LIN {X 0,Y 197.414,Z 518.474,A -85,B 0,C 180,E1 1852.576,E2 1852.576} C_VEL
LIN {X 0,Y 195.678,Z 514.647,A -85,B 0,C 180,E1 1845.984,E2 1845.984} C_VEL
LIN {X 0,Y 194.931,Z 514.01,A -85,B 0,C 180,E1 1839.244,E2 1839.244} C_VEL
LIN {X 0,Y 195.748,Z 514.716,A -85,B 0,C 180,E1 1832.022,E2 1832.022} C_VEL
LIN {X 0,Y 197.692,Z 519.438,A -85,B 0,C 180,E1 1824.497,E2 1824.497} C_VEL
LIN {X 0,Y 199.785,Z 523.662,A -85,B 0,C 180,E1 1819.811,E2 1819.811} C_VEL
LIN {X 0,Y 202.216,Z 528.549,A -85,B 0,C 180,E1 1815.605,E2 1815.605} C_VEL
LIN {X 0,Y 190.643,Z 578.863,A -85,B 0,C 180,E1 1815.121,E2 1815.121} C_VEL
LIN {X 0,Y 183.364,Z 602.487,A -85,B 0,C 180,E1 1814.882,E2 1814.882} C_VEL
LIN {X 0,Y 173.66,Z 626.987,A -85,B 0,C 180,E1 1814.716,E2 1814.716} C_VEL
LIN {X 0,Y 162.076,Z 650.907,A -85,B 0,C 180,E1 1814.426,E2 1814.426} C_VEL
LIN {X 0,Y 149.405,Z 672.786,A -85,B 0,C 180,E1 1813.999,E2 1813.999} C_VEL
LIN {X 0,Y 135.148,Z 693.676,A -85,B 0,C 180,E1 1813.399,E2 1813.399} C_VEL
LIN {X 0,Y 120.37,Z 712.234,A -85,B 0,C 180,E1 1812.599,E2 1812.599} C_VEL
LIN {X 0,Y 104.563,Z 729.321,A -85,B 0,C 180,E1 1811.473,E2 1811.473} C_VEL
LIN {X 0,Y 87.256,Z 745.402,A -85,B 0,C 180,E1 1809.824,E2 1809.824} C_VEL
LIN {X 0,Y 69.557,Z 759.526,A -85,B 0,C 180,E1 1807.39,E2 1807.39} C_VEL
LIN {X 0,Y 52.081,Z 771.407,A -85,B 0,C 180,E1 1803.53,E2 1803.53} C_VEL
LIN {X 0,Y 34.078,Z 781.783,A -85,B 0,C 180,E1 1795.754,E2 1795.754} C_VEL
LIN {X 0,Y 17.731,Z 790.254,A -85,B 0,C 180,E1 1774.376,E2 1774.376} C_VEL
LIN {X 0,Y 11.425,Z 796.051,A -85,B 0,C 180,E1 1709.95,E2 1709.95} C_VEL
LIN {X 0,Y 11.818,Z 796.617,A -85,B 0,C 180,E1 1700.209,E2 1700.209} C_VEL
LIN {X 0,Y 14.795,Z 798.166,A -85,B 0,C 180,E1 1657.527,E2 1657.527} C_VEL
LIN {X 0,Y 9.219,Z 793.702,A -85,B 0,C 180,E1 1601.102,E2 1601.102} C_VEL
LIN {X 0,Y 18.153,Z 786.818,A -85,B 0,C 180,E1 1537.839,E2 1537.839} C_VEL
LIN {X 0,Y 35.521,Z 777.013,A -85,B 0,C 180,E1 1519.997,E2 1519.997} C_VEL
LIN {X 0,Y 54.697,Z 764.948,A -85,B 0,C 180,E1 1513.005,E2 1513.005} C_VEL
LIN {X 0,Y 72.604,Z 751.86,A -85,B 0,C 180,E1 1509.431,E2 1509.431} C_VEL
LIN {X 0,Y 90.666,Z 736.479,A -85,B 0,C 180,E1 1507.024,E2 1507.024} C_VEL
LIN {X 0,Y 107.146,Z 720.254,A -85,B 0,C 180,E1 1505.379,E2 1505.379} C_VEL
LIN {X 0,Y 123.373,Z 701.747,A -85,B 0,C 180,E1 1504.086,E2 1504.086} C_VEL
LIN {X 0,Y 132.523,Z 689.974,A -85,B 0,C 180,E1 1503.457,E2 1503.457} C_VEL
LIN {X 0,Y 136.821,Z 683.736,A -85,B 0,C 180,E1 1502.763,E2 1502.763} C_VEL
LIN {X 0,Y 146.781,Z 666.497,A -85,B 0,C 180,E1 1499.753,E2 1499.753} C_VEL
LIN {X 0,Y 150.068,Z 660.76,A -85,B 0,C 180,E1 1499.343,E2 1499.343} C_VEL
LIN {X 0,Y 162.241,Z 638.701,A -85,B 0,C 180,E1 1498.929,E2 1498.929} C_VEL
LIN {X 0,Y 172.705,Z 616.198,A -85,B 0,C 180,E1 1498.602,E2 1498.602} C_VEL
LIN {X 0,Y 182.088,Z 591.601,A -85,B 0,C 180,E1 1498.323,E2 1498.323} C_VEL
LIN {X 0,Y 189.755,Z 566.126,A -85,B 0,C 180,E1 1498.101,E2 1498.101} C_VEL
LIN {X 0,Y 197.833,Z 531.198,A -85,B 0,C 180,E1 1497.859,E2 1497.859} C_VEL
LIN {X 0,Y 195.599,Z 526.307,A -85,B 0,C 180,E1 1492.537,E2 1492.537} C_VEL
LIN {X 0,Y 193.851,Z 522.423,A -85,B 0,C 180,E1 1485.795,E2 1485.795} C_VEL
LIN {X 0,Y 193.15,Z 521.811,A -85,B 0,C 180,E1 1479.065,E2 1479.065} C_VEL
LIN {X 0,Y 193.929,Z 522.613,A -85,B 0,C 180,E1 1472.071,E2 1472.071} C_VEL
LIN {X 0,Y 195.706,Z 527.054,A -85,B 0,C 180,E1 1464.924,E2 1464.924} C_VEL
LIN {X 0,Y 197.708,Z 531.241,A -85,B 0,C 180,E1 1460.264,E2 1460.264} C_VEL
LIN {X 0,Y 198.994,Z 534.087,A -85,B 0,C 180,E1 1457.774,E2 1457.774} C_VEL
LIN {X 0,Y 188.414,Z 579.035,A -85,B 0,C 180,E1 1457.449,E2 1457.449} C_VEL
LIN {X 0,Y 181.163,Z 602.307,A -85,B 0,C 180,E1 1457.304,E2 1457.304} C_VEL
LIN {X 0,Y 171.68,Z 626.174,A -85,B 0,C 180,E1 1457.274,E2 1457.274} C_VEL
LIN {X 0,Y 160.099,Z 650.057,A -85,B 0,C 180,E1 1457.167,E2 1457.167} C_VEL
LIN {X 0,Y 147.264,Z 672.137,A -85,B 0,C 180,E1 1456.969,E2 1456.969} C_VEL
LIN {X 0,Y 133.065,Z 692.712,A -85,B 0,C 180,E1 1456.673,E2 1456.673} C_VEL
LIN {X 0,Y 118.735,Z 710.564,A -85,B 0,C 180,E1 1456.283,E2 1456.283} C_VEL
LIN {X 0,Y 102.284,Z 728.281,A -85,B 0,C 180,E1 1455.686,E2 1455.686} C_VEL
LIN {X 0,Y 84.816,Z 744.397,A -85,B 0,C 180,E1 1454.865,E2 1454.865} C_VEL
LIN {X 0,Y 67.933,Z 757.735,A -85,B 0,C 180,E1 1453.773,E2 1453.773} C_VEL
LIN {X 0,Y 50.078,Z 769.624,A -85,B 0,C 180,E1 1452.007,E2 1452.007} C_VEL
LIN {X 0,Y 30.308,Z 780.674,A -85,B 0,C 180,E1 1448.365,E2 1448.365} C_VEL
LIN {X 0,Y 12.995,Z 788.665,A -85,B 0,C 180,E1 1438.177,E2 1438.177} C_VEL
LIN {X 0,Y 4.365,Z 794.222,A -85,B 0,C 180,E1 1322.59,E2 1322.59} C_VEL
LIN {X 0,Y 4.321,Z 794.234,A -85,B 0,C 180,E1 1315.544,E2 1315.544} C_VEL
LIN {X 0,Y 8.811,Z 788.86,A -85,B 0,C 180,E1 1156.948,E2 1156.948} C_VEL
LIN {X 0,Y 27.983,Z 779.327,A -85,B 0,C 180,E1 1148.202,E2 1148.202} C_VEL
LIN {X 0,Y 46.158,Z 768.699,A -85,B 0,C 180,E1 1145.432,E2 1145.432} C_VEL
LIN {X 0,Y 65.276,Z 755.458,A -85,B 0,C 180,E1 1143.638,E2 1143.638} C_VEL
LIN {X 0,Y 83.49,Z 740.749,A -85,B 0,C 180,E1 1142.378,E2 1142.378} C_VEL
LIN {X 0,Y 100.753,Z 724.51,A -85,B 0,C 180,E1 1141.414,E2 1141.414} C_VEL
LIN {X 0,Y 116.998,Z 706.864,A -85,B 0,C 180,E1 1140.639,E2 1140.639} C_VEL
LIN {X 0,Y 132.779,Z 686.918,A -85,B 0,C 180,E1 1139.98,E2 1139.98} C_VEL
LIN {X 0,Y 146.231,Z 667.041,A -85,B 0,C 180,E1 1139.476,E2 1139.476} C_VEL
LIN {X 0,Y 150.068,Z 660.76,A -85,B 0,C 180,E1 1139.343,E2 1139.343} C_VEL
LIN {X 0,Y 153.729,Z 654.207,A -85,B 0,C 180,E1 1138.842,E2 1138.842} C_VEL
LIN {X 0,Y 162.215,Z 635.803,A -85,B 0,C 180,E1 1136.382,E2 1136.382} C_VEL
LIN {X 0,Y 165.007,Z 629.769,A -85,B 0,C 180,E1 1136.081,E2 1136.081} C_VEL
LIN {X 0,Y 175.459,Z 605.484,A -85,B 0,C 180,E1 1135.917,E2 1135.917} C_VEL
LIN {X 0,Y 184.182,Z 580.142,A -85,B 0,C 180,E1 1135.777,E2 1135.777} C_VEL
LIN {X 0,Y 191.07,Z 554.146,A -85,B 0,C 180,E1 1135.68,E2 1135.68} C_VEL
LIN {X 0,Y 194.927,Z 536.894,A -85,B 0,C 180,E1 1135.566,E2 1135.566} C_VEL
LIN {X 0,Y 193.45,Z 533.708,A -85,B 0,C 180,E1 1131.672,E2 1131.672} C_VEL
LIN {X 0,Y 192.007,Z 530.188,A -85,B 0,C 180,E1 1125.506,E2 1125.506} C_VEL
LIN {X 0,Y 191.371,Z 529.622,A -85,B 0,C 180,E1 1118.82,E2 1118.82} C_VEL
LIN {X 0,Y 192.091,Z 530.439,A -85,B 0,C 180,E1 1112.238,E2 1112.238} C_VEL
LIN {X 0,Y 193.731,Z 534.669,A -85,B 0,C 180,E1 1105.359,E2 1105.359} C_VEL
LIN {X 0,Y 195.639,Z 538.806,A -85,B 0,C 180,E1 1100.739,E2 1100.739} C_VEL
LIN {X 0,Y 195.909,Z 539.823,A -85,B 0,C 180,E1 1100.007,E2 1100.007} C_VEL
LIN {X 0,Y 186.521,Z 579.131,A -85,B 0,C 180,E1 1099.829,E2 1099.829} C_VEL
LIN {X 0,Y 179.292,Z 602.117,A -85,B 0,C 180,E1 1099.78,E2 1099.78} C_VEL
LIN {X 0,Y 170.102,Z 625.075,A -85,B 0,C 180,E1 1099.88,E2 1099.88} C_VEL
LIN {X 0,Y 159.014,Z 647.884,A -85,B 0,C 180,E1 1099.955,E2 1099.955} C_VEL
LIN {X 0,Y 146.817,Z 668.997,A -85,B 0,C 180,E1 1099.993,E2 1099.993} C_VEL
LIN {X 0,Y 133.013,Z 689.374,A -85,B 0,C 180,E1 1100.026,E2 1100.026} C_VEL
LIN {X 0,Y 117.599,Z 708.853,A -85,B 0,C 180,E1 1100.049,E2 1100.049} C_VEL
LIN {X 0,Y 101.988,Z 725.805,A -85,B 0,C 180,E1 1100.059,E2 1100.059} C_VEL
LIN {X 0,Y 85.184,Z 741.471,A -85,B 0,C 180,E1 1100.136,E2 1100.136} C_VEL
LIN {X 0,Y 67.173,Z 755.75,A -85,B 0,C 180,E1 1100.35,E2 1100.35} C_VEL
LIN {X 0,Y 49.246,Z 767.828,A -85,B 0,C 180,E1 1100.973,E2 1100.973} C_VEL
LIN {X 0,Y 30.612,Z 778.351,A -85,B 0,C 180,E1 1103.048,E2 1103.048} C_VEL
LIN {X 0,Y 12.717,Z 786.715,A -85,B 0,C 180,E1 1113.319,E2 1113.319} C_VEL
LIN {X 0,Y 12.158,Z 786.943,A -85,B 0,C 180,E1 1115.067,E2 1115.067} C_VEL
LIN {X 0,Y 27.951,Z 778.436,A -85,B 0,C 180,E1 1131.857,E2 1131.857} C_VEL
LIN {X 0,Y 47.934,Z 766.344,A -85,B 0,C 180,E1 1135.737,E2 1135.737} C_VEL
LIN {X 0,Y 65.8,Z 753.744,A -85,B 0,C 180,E1 1136.67,E2 1136.67} C_VEL
LIN {X 0,Y 84.699,Z 738.08,A -85,B 0,C 180,E1 1136.925,E2 1136.925} C_VEL
LIN {X 0,Y 101.794,Z 721.638,A -85,B 0,C 180,E1 1136.885,E2 1136.885} C_VEL
LIN {X 0,Y 118.47,Z 702.955,A -85,B 0,C 180,E1 1136.736,E2 1136.736} C_VEL
LIN {X 0,Y 134.22,Z 682.356,A -85,B 0,C 180,E1 1136.534,E2 1136.534} C_VEL
LIN {X 0,Y 147.907,Z 661.457,A -85,B 0,C 180,E1 1136.341,E2 1136.341} C_VEL
LIN {X 0,Y 160.095,Z 639.643,A -85,B 0,C 180,E1 1136.154,E2 1136.154} C_VEL
LIN {X 0,Y 165.007,Z 629.769,A -85,B 0,C 180,E1 1136.081,E2 1136.081} C_VEL
LIN {X 0,Y 168.047,Z 622.718,A -85,B 0,C 180,E1 1135.702,E2 1135.702} C_VEL
LIN {X 0,Y 174.846,Z 603.563,A -85,B 0,C 180,E1 1133.617,E2 1133.617} C_VEL
LIN {X 0,Y 176.978,Z 597.31,A -85,B 0,C 180,E1 1133.331,E2 1133.331} C_VEL
LIN {X 0,Y 184.885,Z 572.665,A -85,B 0,C 180,E1 1133.322,E2 1133.322} C_VEL
LIN {X 0,Y 192.203,Z 542.924,A -85,B 0,C 180,E1 1133.26,E2 1133.26} C_VEL
LIN {X 0,Y 191.224,Z 540.862,A -85,B 0,C 180,E1 1130.369,E2 1130.369} C_VEL
LIN {X 0,Y 190.25,Z 538.003,A -85,B 0,C 180,E1 1125.615,E2 1125.615} C_VEL
LIN {X 0,Y 189.59,Z 537.433,A -85,B 0,C 180,E1 1118.697,E2 1118.697} C_VEL
LIN {X 0,Y 190.244,Z 538.258,A -85,B 0,C 180,E1 1112.411,E2 1112.411} C_VEL
LIN {X 0,Y 191.767,Z 542.284,A -85,B 0,C 180,E1 1105.803,E2 1105.803} C_VEL
LIN {X 0,Y 193.046,Z 545.384,A -85,B 0,C 180,E1 1102.303,E2 1102.303} C_VEL
LIN {X 0,Y 184.537,Z 580.024,A -85,B 0,C 180,E1 1102.241,E2 1102.241} C_VEL
LIN {X 0,Y 177.216,Z 602.742,A -85,B 0,C 180,E1 1102.298,E2 1102.298} C_VEL
LIN {X 0,Y 167.786,Z 626.038,A -85,B 0,C 180,E1 1102.543,E2 1102.543} C_VEL
LIN {X 0,Y 156.717,Z 648.632,A -85,B 0,C 180,E1 1102.804,E2 1102.804} C_VEL
LIN {X 0,Y 143.487,Z 671.222,A -85,B 0,C 180,E1 1103.113,E2 1103.113} C_VEL
LIN {X 0,Y 130.284,Z 690.272,A -85,B 0,C 180,E1 1103.452,E2 1103.452} C_VEL
LIN {X 0,Y 115.374,Z 708.818,A -85,B 0,C 180,E1 1103.909,E2 1103.909} C_VEL
LIN {X 0,Y 98.487,Z 726.872,A -85,B 0,C 180,E1 1104.588,E2 1104.588} C_VEL
LIN {X 0,Y 82.024,Z 742.026,A -85,B 0,C 180,E1 1105.59,E2 1105.59} C_VEL
LIN {X 0,Y 65.601,Z 755.006,A -85,B 0,C 180,E1 1107.196,E2 1107.196} C_VEL
LIN {X 0,Y 47.568,Z 767.184,A -85,B 0,C 180,E1 1110.505,E2 1110.505} C_VEL
LIN {X 0,Y 31.392,Z 776.705,A -85,B 0,C 180,E1 1117.827,E2 1117.827} C_VEL
LIN {X 0,Y 49.531,Z 764.811,A -85,B 0,C 180,E1 1126.587,E2 1126.587} C_VEL
LIN {X 0,Y 68.55,Z 750.724,A -85,B 0,C 180,E1 1130.087,E2 1130.087} C_VEL
LIN {X 0,Y 85.458,Z 736.323,A -85,B 0,C 180,E1 1131.603,E2 1131.603} C_VEL
LIN {X 0,Y 102.702,Z 719.32,A -85,B 0,C 180,E1 1132.453,E2 1132.453} C_VEL
LIN {X 0,Y 119.053,Z 700.615,A -85,B 0,C 180,E1 1132.912,E2 1132.912} C_VEL
LIN {X 0,Y 133.689,Z 681.228,A -85,B 0,C 180,E1 1133.143,E2 1133.143} C_VEL
LIN {X 0,Y 147.653,Z 659.548,A -85,B 0,C 180,E1 1133.27,E2 1133.27} C_VEL
LIN {X 0,Y 159.974,Z 636.991,A -85,B 0,C 180,E1 1133.319,E2 1133.319} C_VEL
LIN {X 0,Y 170.786,Z 613.308,A -85,B 0,C 180,E1 1133.338,E2 1133.338} C_VEL
LIN {X 0,Y 176.978,Z 597.31,A -85,B 0,C 180,E1 1133.331,E2 1133.331} C_VEL
LIN {X 0,Y 179.399,Z 590.013,A -85,B 0,C 180,E1 1133.015,E2 1133.015} C_VEL
LIN {X 0,Y 184.493,Z 570.266,A -85,B 0,C 180,E1 1131.105,E2 1131.105} C_VEL
LIN {X 0,Y 186.05,Z 563.821,A -85,B 0,C 180,E1 1130.885,E2 1130.885} C_VEL
LIN {X 0,Y 189.595,Z 549.036,A -85,B 0,C 180,E1 1130.916,E2 1130.916} C_VEL
LIN {X 0,Y 188.366,Z 545.739,A -85,B 0,C 180,E1 1125.097,E2 1125.097} C_VEL
LIN {X 0,Y 187.838,Z 545.283,A -85,B 0,C 180,E1 1118.025,E2 1118.025} C_VEL
LIN {X 0,Y 188.399,Z 546.073,A -85,B 0,C 180,E1 1112.588,E2 1112.588} C_VEL
LIN {X 0,Y 189.857,Z 550.046,A -85,B 0,C 180,E1 1106.082,E2 1106.082} C_VEL
LIN {X 0,Y 190.247,Z 551.357,A -85,B 0,C 180,E1 1104.657,E2 1104.657} C_VEL
LIN {X 0,Y 182.568,Z 581.762,A -85,B 0,C 180,E1 1104.702,E2 1104.702} C_VEL
LIN {X 0,Y 174.968,Z 604.694,A -85,B 0,C 180,E1 1104.891,E2 1104.891} C_VEL
LIN {X 0,Y 165.84,Z 626.92,A -85,B 0,C 180,E1 1105.272,E2 1105.272} C_VEL
LIN {X 0,Y 154.807,Z 649.12,A -85,B 0,C 180,E1 1105.721,E2 1105.721} C_VEL
LIN {X 0,Y 141.634,Z 671.367,A -85,B 0,C 180,E1 1106.302,E2 1106.302} C_VEL
LIN {X 0,Y 126.864,Z 692.488,A -85,B 0,C 180,E1 1107.064,E2 1107.064} C_VEL
LIN {X 0,Y 111.054,Z 711.76,A -85,B 0,C 180,E1 1108.088,E2 1108.088} C_VEL
LIN {X 0,Y 96.34,Z 727.19,A -85,B 0,C 180,E1 1109.346,E2 1109.346} C_VEL
LIN {X 0,Y 78.614,Z 743.277,A -85,B 0,C 180,E1 1111.569,E2 1111.569} C_VEL
LIN {X 0,Y 61.191,Z 756.944,A -85,B 0,C 180,E1 1115.232,E2 1115.232} C_VEL
LIN {X 0,Y 52.488,Z 763.095,A -85,B 0,C 180,E1 1118.29,E2 1118.29} C_VEL
LIN {X 0,Y 69.615,Z 749.626,A -85,B 0,C 180,E1 1123.566,E2 1123.566} C_VEL
LIN {X 0,Y 87.501,Z 733.772,A -85,B 0,C 180,E1 1126.505,E2 1126.505} C_VEL
LIN {X 0,Y 104.245,Z 716.765,A -85,B 0,C 180,E1 1128.138,E2 1128.138} C_VEL
LIN {X 0,Y 119.591,Z 698.78,A -85,B 0,C 180,E1 1129.121,E2 1129.121} C_VEL
LIN {X 0,Y 134.828,Z 678.056,A -85,B 0,C 180,E1 1129.792,E2 1129.792} C_VEL
LIN {X 0,Y 148.423,Z 656.428,A -85,B 0,C 180,E1 1130.216,E2 1130.216} C_VEL
LIN {X 0,Y 160.283,Z 634.216,A -85,B 0,C 180,E1 1130.49,E2 1130.49} C_VEL
LIN {X 0,Y 170.578,Z 611.086,A -85,B 0,C 180,E1 1130.681,E2 1130.681} C_VEL
LIN {X 0,Y 179.309,Z 587.092,A -85,B 0,C 180,E1 1130.804,E2 1130.804} C_VEL
LIN {X 0,Y 186.05,Z 563.821,A -85,B 0,C 180,E1 1130.885,E2 1130.885} C_VEL
LIN {X 0,Y 186.666,Z 560.864,A -85,B 0,C 180,E1 1130.595,E2 1130.595} C_VEL
LIN {X 0,Y 187.051,Z 557.972,A -85,B 0,C 180,E1 1129.734,E2 1129.734} C_VEL
LIN {X 0,Y 187.086,Z 555.546,A -85,B 0,C 180,E1 1128.236,E2 1128.236} C_VEL
LIN {X 0,Y 186.663,Z 553.75,A -85,B 0,C 180,E1 1125.585,E2 1125.585} C_VEL
LIN {X 0,Y 186.449,Z 553.431,A -85,B 0,C 180,E1 1124.227,E2 1124.227} C_VEL
LIN {X 0,Y 186.088,Z 553.11,A -85,B 0,C 180,E1 1117.331,E2 1117.331} C_VEL
LIN {X 0,Y 186.533,Z 553.764,A -85,B 0,C 180,E1 1112.955,E2 1112.955} C_VEL
LIN {X 0,Y 187.732,Z 557.193,A -85,B 0,C 180,E1 1107.079,E2 1107.079} C_VEL
LIN {X 0,Y 180.946,Z 583.054,A -85,B 0,C 180,E1 1107.206,E2 1107.206} C_VEL
LIN {X 0,Y 173.287,Z 605.613,A -85,B 0,C 180,E1 1107.519,E2 1107.519} C_VEL
LIN {X 0,Y 163.2,Z 629.567,A -85,B 0,C 180,E1 1108.097,E2 1108.097} C_VEL
LIN {X 0,Y 151.488,Z 652.549,A -85,B 0,C 180,E1 1108.798,E2 1108.798} C_VEL
LIN {X 0,Y 138.654,Z 673.782,A -85,B 0,C 180,E1 1109.673,E2 1109.673} C_VEL
LIN {X 0,Y 125.146,Z 692.94,A -85,B 0,C 180,E1 1110.745,E2 1110.745} C_VEL
LIN {X 0,Y 109.95,Z 711.427,A -85,B 0,C 180,E1 1112.262,E2 1112.262} C_VEL
LIN {X 0,Y 94.434,Z 727.732,A -85,B 0,C 180,E1 1114.337,E2 1114.337} C_VEL
LIN {X 0,Y 78.146,Z 742.722,A -85,B 0,C 180,E1 1117.52,E2 1117.52} C_VEL
LIN {X 0,Y 75.156,Z 745.279,A -85,B 0,C 180,E1 1118.378,E2 1118.378} C_VEL
LIN {X 0,Y 91.926,Z 729.428,A -85,B 0,C 180,E1 1121.971,E2 1121.971} C_VEL
LIN {X 0,Y 108.899,Z 711.075,A -85,B 0,C 180,E1 1124.27,E2 1124.27} C_VEL
LIN {X 0,Y 123.793,Z 692.576,A -85,B 0,C 180,E1 1125.646,E2 1125.646} C_VEL
LIN {X 0,Y 137.611,Z 672.748,A -85,B 0,C 180,E1 1126.591,E2 1126.591} C_VEL
LIN {X 0,Y 151.038,Z 650.271,A -85,B 0,C 180,E1 1127.282,E2 1127.282} C_VEL
LIN {X 0,Y 162.505,Z 627.566,A -85,B 0,C 180,E1 1127.756,E2 1127.756} C_VEL
LIN {X 0,Y 172.07,Z 604.937,A -85,B 0,C 180,E1 1128.074,E2 1128.074} C_VEL
LIN {X 0,Y 180.513,Z 580.378,A -85,B 0,C 180,E1 1128.306,E2 1128.306} C_VEL
LIN {X 0,Y 187.165,Z 555.546,A -85,B 0,C 180,E1 1128.465,E2 1128.465} C_VEL
LIN {X 0,Y 186.565,Z 553.526,A -85,B 0,C 180,E1 1124.979,E2 1124.979} C_VEL
LIN {X 0,Y 186.449,Z 553.431,A -85,B 0,C 180,E1 1124.227,E2 1124.227} C_VEL
LIN {X 0,Y 185.967,Z 554.06,A -85,B 0,C 180,E1 1121.683,E2 1121.683} C_VEL
LIN {X 0,Y 185.069,Z 557.52,A -85,B 0,C 180,E1 1117.688,E2 1117.688} C_VEL
LIN {X 0,Y 184.642,Z 561.35,A -85,B 0,C 180,E1 1113.482,E2 1113.482} C_VEL
LIN {X 0,Y 185.11,Z 563.874,A -85,B 0,C 180,E1 1109.553,E2 1109.553} C_VEL
LIN {X 0,Y 178.561,Z 587.509,A -85,B 0,C 180,E1 1109.789,E2 1109.789} C_VEL
LIN {X 0,Y 170.75,Z 609.585,A -85,B 0,C 180,E1 1110.272,E2 1110.272} C_VEL
LIN {X 0,Y 160.971,Z 632.201,A -85,B 0,C 180,E1 1111.007,E2 1111.007} C_VEL
LIN {X 0,Y 150.107,Z 653.169,A -85,B 0,C 180,E1 1111.876,E2 1111.876} C_VEL
LIN {X 0,Y 137.179,Z 674.373,A -85,B 0,C 180,E1 1113.058,E2 1113.058} C_VEL
LIN {X 0,Y 123.35,Z 693.875,A -85,B 0,C 180,E1 1114.561,E2 1114.561} C_VEL
LIN {X 0,Y 108.407,Z 712.154,A -85,B 0,C 180,E1 1116.649,E2 1116.649} C_VEL
LIN {X 0,Y 99.125,Z 722.266,A -85,B 0,C 180,E1 1118.33,E2 1118.33} C_VEL
LIN {X 0,Y 114.683,Z 704.055,A -85,B 0,C 180,E1 1120.825,E2 1120.825} C_VEL
LIN {X 0,Y 129.608,Z 684.108,A -85,B 0,C 180,E1 1122.539,E2 1122.539} C_VEL
LIN {X 0,Y 143.603,Z 662.462,A -85,B 0,C 180,E1 1123.742,E2 1123.742} C_VEL
LIN {X 0,Y 155.761,Z 640.448,A -85,B 0,C 180,E1 1124.565,E2 1124.565} C_VEL
LIN {X 0,Y 166.373,Z 617.505,A -85,B 0,C 180,E1 1125.158,E2 1125.158} C_VEL
LIN {X 0,Y 175.39,Z 593.95,A -85,B 0,C 180,E1 1125.587,E2 1125.587} C_VEL
LIN {X 0,Y 183.08,Z 568.73,A -85,B 0,C 180,E1 1125.91,E2 1125.91} C_VEL
LIN {X 0,Y 184.784,Z 561.906,A -85,B 0,C 180,E1 1125.953,E2 1125.953} C_VEL
LIN {X 0,Y 184.594,Z 561.21,A -85,B 0,C 180,E1 1124.157,E2 1124.157} C_VEL
LIN {X 0,Y 184.28,Z 560.906,A -85,B 0,C 180,E1 1117.026,E2 1117.026} C_VEL
LIN {X 0,Y 184.642,Z 561.35,A -85,B 0,C 180,E1 1113.482,E2 1113.482} C_VEL
LIN {X 0,Y 184.501,Z 562.678,A -85,B 0,C 180,E1 1112.765,E2 1112.765} C_VEL
LIN {X 0,Y 183.956,Z 565.591,A -85,B 0,C 180,E1 1112.183,E2 1112.183} C_VEL
LIN {X 0,Y 182.791,Z 570.552,A -85,B 0,C 180,E1 1111.875,E2 1111.875} C_VEL
LIN {X 0,Y 178.799,Z 584.325,A -85,B 0,C 180,E1 1112.301,E2 1112.301} C_VEL
LIN {X 0,Y 171.365,Z 605.839,A -85,B 0,C 180,E1 1112.847,E2 1112.847} C_VEL
LIN {X 0,Y 161.689,Z 628.835,A -85,B 0,C 180,E1 1113.731,E2 1113.731} C_VEL
LIN {X 0,Y 149.937,Z 652.043,A -85,B 0,C 180,E1 1114.9,E2 1114.9} C_VEL
LIN {X 0,Y 137.211,Z 673.284,A -85,B 0,C 180,E1 1116.369,E2 1116.369} C_VEL
LIN {X 0,Y 124.15,Z 692.123,A -85,B 0,C 180,E1 1118.208,E2 1118.208} C_VEL
LIN {X 0,Y 137.997,Z 671.492,A -85,B 0,C 180,E1 1119.955,E2 1119.955} C_VEL
LIN {X 0,Y 150.345,Z 650.239,A -85,B 0,C 180,E1 1121.169,E2 1121.169} C_VEL
LIN {X 0,Y 162.032,Z 626.576,A -85,B 0,C 180,E1 1122.117,E2 1122.117} C_VEL
LIN {X 0,Y 171.87,Z 602.569,A -85,B 0,C 180,E1 1122.78,E2 1122.78} C_VEL
LIN {X 0,Y 180.266,Z 577.125,A -85,B 0,C 180,E1 1123.269,E2 1123.269} C_VEL
LIN {X 0,Y 182.584,Z 568.874,A -85,B 0,C 180,E1 1123.335,E2 1123.335} C_VEL
LIN {X 0,Y 182.361,Z 568.683,A -85,B 0,C 180,E1 1116.694,E2 1116.694} C_VEL
LIN {X 0,Y 182.685,Z 569.323,A -85,B 0,C 180,E1 1113.364,E2 1113.364} C_VEL
LIN {X 0,Y 182.787,Z 570.299,A -85,B 0,C 180,E1 1112.101,E2 1112.101} C_VEL
LIN {X 0,Y 178.799,Z 584.325,A -85,B 0,C 180,E1 1112.301,E2 1112.301} C_VEL
LIN {X 0,Y 176.455,Z 591.577,A -85,B 0,C 180,E1 1112.766,E2 1112.766} C_VEL
LIN {X 0,Y 168.905,Z 610.92,A -85,B 0,C 180,E1 1115.576,E2 1115.576} C_VEL
LIN {X 0,Y 166.801,Z 615.961,A -85,B 0,C 180,E1 1115.972,E2 1115.972} C_VEL
LIN {X 0,Y 156.233,Z 639.264,A -85,B 0,C 180,E1 1117.184,E2 1117.184} C_VEL
LIN {X 0,Y 149.682,Z 651.809,A -85,B 0,C 180,E1 1118.011,E2 1118.011} C_VEL
LIN {X 0,Y 160.884,Z 629.07,A -85,B 0,C 180,E1 1119.167,E2 1119.167} C_VEL
LIN {X 0,Y 170.567,Z 605.611,A -85,B 0,C 180,E1 1120.015,E2 1120.015} C_VEL
LIN {X 0,Y 178.751,Z 581.287,A -85,B 0,C 180,E1 1120.633,E2 1120.633} C_VEL
LIN {X 0,Y 180.17,Z 576.343,A -85,B 0,C 180,E1 1120.7,E2 1120.7} C_VEL
LIN {X 0,Y 180.419,Z 576.707,A -85,B 0,C 180,E1 1114.717,E2 1114.717} C_VEL
LIN {X 0,Y 173.253,Z 599.245,A -85,B 0,C 180,E1 1115.288,E2 1115.288} C_VEL
LIN {X 0,Y 166.801,Z 615.961,A -85,B 0,C 180,E1 1115.972,E2 1115.972} C_VEL
LIN {X 0,Y 167.136,Z 615.063,A -85,B 0,C 180,E1 1116.38,E2 1116.38} C_VEL
LIN {X 0,Y 169.455,Z 609.127,A -85,B 0,C 180,E1 1117.03,E2 1117.03} C_VEL
LIN {X 0,Y 175.071,Z 593.377,A -85,B 0,C 180,E1 1117.53,E2 1117.53} C_VEL
LIN {X 0,Y 177.83,Z 584.796,A -85,B 0,C 180,E1 1117.463,E2 1117.463} C_VEL
LIN {X 0,Y 178.047,Z 584.073,A -85,B 0,C 180,E1 1117.51,E2 1117.51} C_VEL
LIN {X 0,Y 177.955,Z 584.267,A -85,B 0,C 180,E1 1117.988,E2 1117.988} C_VEL
LIN {X 0,Y 175.155,Z 592.987,A -85,B 0,C 180,E1 1117.716,E2 1117.716} C_VEL
LIN {X 0,Y 177.83,Z 584.796,A -85,B 0,C 180,E1 1117.463,E2 1117.463} C_VEL
LIN {X 0,Y 181.6,Z 585.427,A -85,B 0,C 180,E1 1117.148,E2 1117.148} C_VEL
LIN {X 0,Y 181.6,Z 862.5,A -85,B 0,C 180,E1 1117.148,E2 1117.148} C_VEL
LIN {X 0,Y 181.6,Z 862.5,A -85,B 0,C 180,E1 1117.148,E2 1117.148}

QRS_NEXT_CUT()

QRS_NEXT()
QRS_HOME()

END
